Fanuc KAREL source: NC0077.KL

-- PROVISIONAL review KL for V770-1; original PC SHA256 d4ef4ff7c86d51b0b43562d0b308ac87531fa4fa4375003eec740a43f32a0a59
-- Incomplete behavior may be omitted. Consult companion uncertainty JSON. Do not deploy.
PROGRAM NC0077
%NOLOCKGROUP
-- UNRESOLVED_LOCAL_POOL 1 cells at code offset 3; source declarations unknown
-- DIRECT_LOCAL_WORD_ACCESS alone does not prove INTEGER, REAL, or BOOLEAN
BEGIN
  -- UNRESOLVED_PC offsets 0-8; opcodes 2B,2C,7B
  -- UNRESOLVED_PC offsets 13-20; opcodes 9D,23
  -- UNRESOLVED_PC offsets 25-42; opcodes 21,2E,59,79
  -- UNRESOLVED_PC offsets 47-64; opcodes 21,2E,59,79
  -- UNRESOLVED_PC offsets 69-86; opcodes 21,2E,59,79
  -- UNRESOLVED_PC offsets 91-108; opcodes 21,2E,59,79
  -- UNRESOLVED_PC offsets 113-130; opcodes 21,2E,59,79
  -- UNRESOLVED_PC offsets 135-152; opcodes 21,2E,59,79
  -- UNRESOLVED_PC offsets 157-174; opcodes 21,2E,59,79
  -- UNRESOLVED_PC offsets 179-196; opcodes 21,2E,59,79
  -- UNRESOLVED_PC offsets 201-218; opcodes 21,2E,59,79
  -- UNRESOLVED_PC offsets 223-240; opcodes 21,2E,59,79
  -- UNRESOLVED_PC offsets 245-259; opcodes 21,9D,52,23
  -- UNRESOLVED_PC offsets 264-269; opcodes 7A
  -- UNRESOLVED_PC offsets 274-279; opcodes 7A
  -- UNRESOLVED_PC offsets 284-289; opcodes 7A
  -- UNRESOLVED_PC offsets 294-299; opcodes 7A
  -- UNRESOLVED_PC offsets 304-309; opcodes 7A
  -- UNRESOLVED_PC offsets 314-319; opcodes 7A
  -- UNRESOLVED_PC offsets 324-329; opcodes 7A
  -- UNRESOLVED_PC offsets 334-339; opcodes 7A
  -- UNRESOLVED_PC offsets 344-349; opcodes 7A
  -- UNRESOLVED_PC offsets 354-359; opcodes 7A
  -- UNRESOLVED_PC offsets 364-368; opcodes 7F
  -- UNRESOLVED_PC offsets 373-377; opcodes 27,AA
  -- UNRESOLVED_PC offsets 382-386; opcodes 7F
END NC0077
